{attribute addProperty BoxType "EK1100-0000-0018"}
{attribute addProperty Id "Beckhoff_EL47xxEK1122Beckhoff_EL47xxEK1122_4AFA0311162A_0001_EL4712_0000_0000EL4712_C8B4D13D44055A_0002_EL4712_0000_0001EL4712_C8B4D13D44055A_0003_EL4732_0001_0000EL4732_13EEB3C313617A_0004_EL4732_0000_0002EL4732_C8B4D13D44055A_0005_EL4732_0000_0003EL4732_C8B4D13D44055A_0006_EL4732_0000_0004EL4732_C8B4D13D44055"}
{attribute addProperty CRC "2905781578"}
{attribute addProperty SizeInBites "2352"}
{attribute addProperty SizeInBytes "294"}
TYPE Beckhoff_EL47xx_AD32B54A EXTENDS EK1100_179A0949 :
STRUCT
	{attribute addProperty Name "Beckhoff_EL47xxEK1122"}
	Beckhoff_EL47xxEK1122 : Beckhoff_EL47xxEK1122_4AFA0311;
	{attribute addProperty Name "A_0001_EL4712_0000_0000"}
	A_0001_EL4712_0000_0000 : EL4712_C8B4D13D;
	{attribute addProperty Name "A_0002_EL4712_0000_0001"}
	A_0002_EL4712_0000_0001 : EL4712_C8B4D13D;
	{attribute addProperty Name "A_0003_EL4732_0001_0000"}
	A_0003_EL4732_0001_0000 : EL4732_13EEB3C3;
	{attribute addProperty Name "A_0004_EL4732_0000_0002"}
	A_0004_EL4732_0000_0002 : EL4732_C8B4D13D;
	{attribute addProperty Name "A_0005_EL4732_0000_0003"}
	A_0005_EL4732_0000_0003 : EL4732_C8B4D13D;
	{attribute addProperty Name "A_0006_EL4732_0000_0004"}
	A_0006_EL4732_0000_0004 : EL4732_C8B4D13D;
END_STRUCT
END_TYPE

(* stored: Version 1.2.0.0, ProductVersion 3.1.4024.9
   DUT Beckhoff_EL47xx_AD32B54A: Id {ecd43f67-7cca-41cc-acf6-e103a977f42b} *)
